(* PLC project Beremiz SVGUI Test, beremiz Beremiz 0.0 *)
(* stored: creationDateTime 2008-12-14T16:21:19, modificationDateTime 2020-06-02T18:02:02 *)

PROGRAM main_pytest
  VAR
    counter : INT;
    Start_Stop : Button;
    Counter_TextCtrl : TextCtrl;
    State_LedCtrl : Led;
  END_VAR
  VAR  (* added by the conversion: wires and edge detectors of the diagram *)
    _AND96_OUT : BOOL;
    _ADD32_ENO : BOOL;
    _ADD32_OUT : INT;
  END_VAR

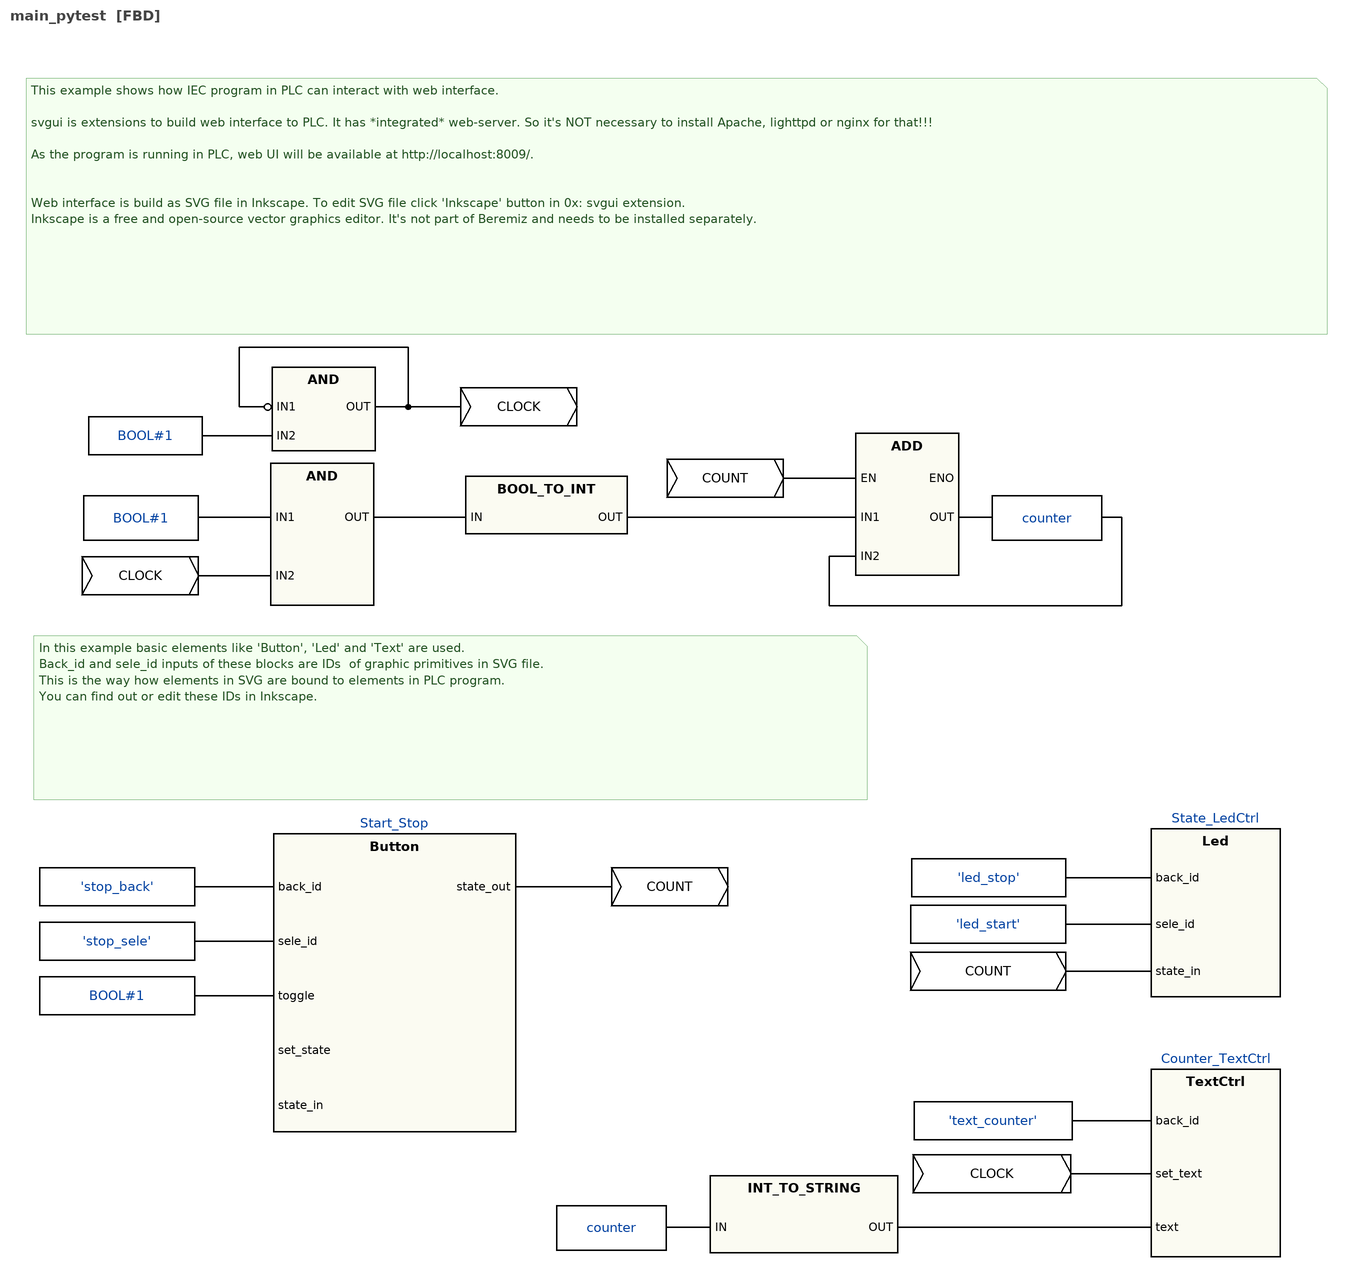
(* FBD diagram, written out as Structured Text *)
(* This example shows how IEC program in PLC can interact with web interface. 

svgui is extensions to build web interface to PLC. It has *integrated* web-server. So it's NOT necessary to install Apache, lighttpd or nginx for that!!!

As the program is running in PLC, web UI will be available at http://localhost:8009/.


Web interface is build as SVG file in Inkscape. To edit SVG file click 'Inkscape' button in 0x: svgui extension. 
Inkscape is a free and open-source vector graphics editor. It's not part of Beremiz and needs to be installed separately. *)
Start_Stop(back_id := 'stop_back', sele_id := 'stop_sele', toggle := BOOL#1);
_AND96_OUT := NOT _AND96_OUT AND BOOL#1;
_ADD32_OUT := ADD(EN := Start_Stop.state_out, IN1 := BOOL_TO_INT(BOOL#1 AND _AND96_OUT), IN2 := counter, ENO => _ADD32_ENO);
IF _ADD32_ENO THEN counter := _ADD32_OUT; END_IF;
(* In this example basic elements like 'Button', 'Led' and 'Text' are used. 
Back_id and sele_id inputs of these blocks are IDs  of graphic primitives in SVG file. 
This is the way how elements in SVG are bound to elements in PLC program. 
You can find out or edit these IDs in Inkscape. *)
State_LedCtrl(back_id := 'led_stop', sele_id := 'led_start', state_in := Start_Stop.state_out);
Counter_TextCtrl(back_id := 'text_counter', set_text := _AND96_OUT, text := INT_TO_STRING(counter));
END_PROGRAM

CONFIGURATION config
  RESOURCE res_pytest ON PLC
    TASK pytest_task(INTERVAL := t#100ms, PRIORITY := 0);
    PROGRAM pytest_instance : main_pytest;
  END_RESOURCE
END_CONFIGURATION
